// Mitsubishi GX Works2 project: PLC_Group2   PLC: FX3G

// global labels: Global1
VAR_GLOBAL
  StartDay AT X007 : BOOL;
  EmergencyButton AT X011 : BOOL;
  SystemOnLight AT Y007 : BOOL;
  YeastStartValue AT D1160 : INT;
  YeastStock AT D1100 : INT;
  MaltStartValue AT D1170 : INT;
  MaltStock AT D1120 : INT;
  HopsStartValue AT D1180 : INT;
  HopsStock AT D1130 : INT;
  StartCooking AT X001 : BOOL;
  BeerTypeNumber AT D1140 : INT;
END_VAR
VAR_GLOBAL CONSTANT
  Const_5 : INT := 5;
END_VAR
VAR_GLOBAL
  LagerChosen AT M1 : BOOL;
END_VAR
VAR_GLOBAL CONSTANT
  Const_6 : INT := 6;
END_VAR
VAR_GLOBAL
  PilsnerChosen AT M2 : BOOL;
END_VAR
VAR_GLOBAL CONSTANT
  Const_400 : INT := 400;
  Const_150 : INT := 150;
  Const_12 : INT := 12;
  Const_60 : INT := 60;
END_VAR
VAR_GLOBAL
  LagerStockExists AT M3 : BOOL;
END_VAR
VAR_GLOBAL CONSTANT
  Const_120 : INT := 120;
  Const_53 : INT := 53;
END_VAR
VAR_GLOBAL
  PilsnerStockExists AT M4 : BOOL;
END_VAR
VAR_GLOBAL CONSTANT
  Const_4 : INT := 4;
END_VAR
VAR_GLOBAL
  CookingLight AT Y001 : BOOL;
END_VAR
VAR_GLOBAL CONSTANT
  Const_4_Seconds : INT := 40;
END_VAR
VAR_GLOBAL
  CookingTimeIsOver AT TS0 : BOOL;
  CookingTime AT TC0 : BOOL;
  BeerTypeInput AT D8280 : INT;
  StartFermentation AT X005 : BOOL;
  LagerFermentationTimer AT TC1 : BOOL;
  PilsnerFermentationTimer AT TC2 : BOOL;
  Lager_F_TimerIsOver AT TS1 : BOOL;
  Pilsner_F_TimerIsOver AT TS2 : BOOL;
  FermentationIsOver AT M5 : BOOL;
  BlinkingLight1 AT TC3 : BOOL;
  BlinkingLight2 AT TC4 : BOOL;
  BlinkingLight2IsOver AT TS4 : BOOL;
  BlinkingHelp AT M6 : BOOL;
  BlinkingLight1IsOver AT TS3 : BOOL;
  BlinkingLightBall1 AT Y003 : BOOL;
  BlinkingLightBall2 AT Y004 : BOOL;
END_VAR
VAR_GLOBAL CONSTANT
  Const_Half_Second : INT := 5;
END_VAR
VAR_GLOBAL
  StartPacking AT X002 : BOOL;
  Count6Bottles AT CC1 : BOOL;
END_VAR
VAR_GLOBAL CONSTANT
  Counter_6 : INT := 6;
END_VAR
VAR_GLOBAL
  PackBottle AT X000 : BOOL;
  Finished6Bottles AT CS1 : BOOL;
  PackingLight AT Y002 : BOOL;
  TotalPacks AT D1150 : INT;
END_VAR
VAR_GLOBAL CONSTANT
  Const_1 : INT := 1;
END_VAR
VAR_GLOBAL
  NoStock AT M7 : BOOL;
  AnalogOutput AT D8282 : INT;
  GotLagerYeast AT M8 : BOOL;
  GotLagerMalt AT M9 : BOOL;
  GotLagerHops AT M10 : BOOL;
  GotPilsnerYeast AT M11 : BOOL;
  GotPilsnerMalt AT M12 : BOOL;
  GotPilsnerHops AT M13 : BOOL;
END_VAR
VAR_GLOBAL CONSTANT
  Const_40 : INT := 40;
  Const_0 : INT;
END_VAR

// task Task_01 (event TRUE, interval 0, priority 31): POU_01

PROGRAM POU_01
VAR
  TS00 : BOOL;
  TC0 : BOOL;
END_VAR
VAR CONSTANT
  Const_3_Seconds : INT := 30;
  Const_10 : REAL := -10;
END_VAR
(* structured ladder/FBD written out as ST: instructions are called as NAME(EN, inputs, outputs); _pN, _eN, _tN stand for wires *)
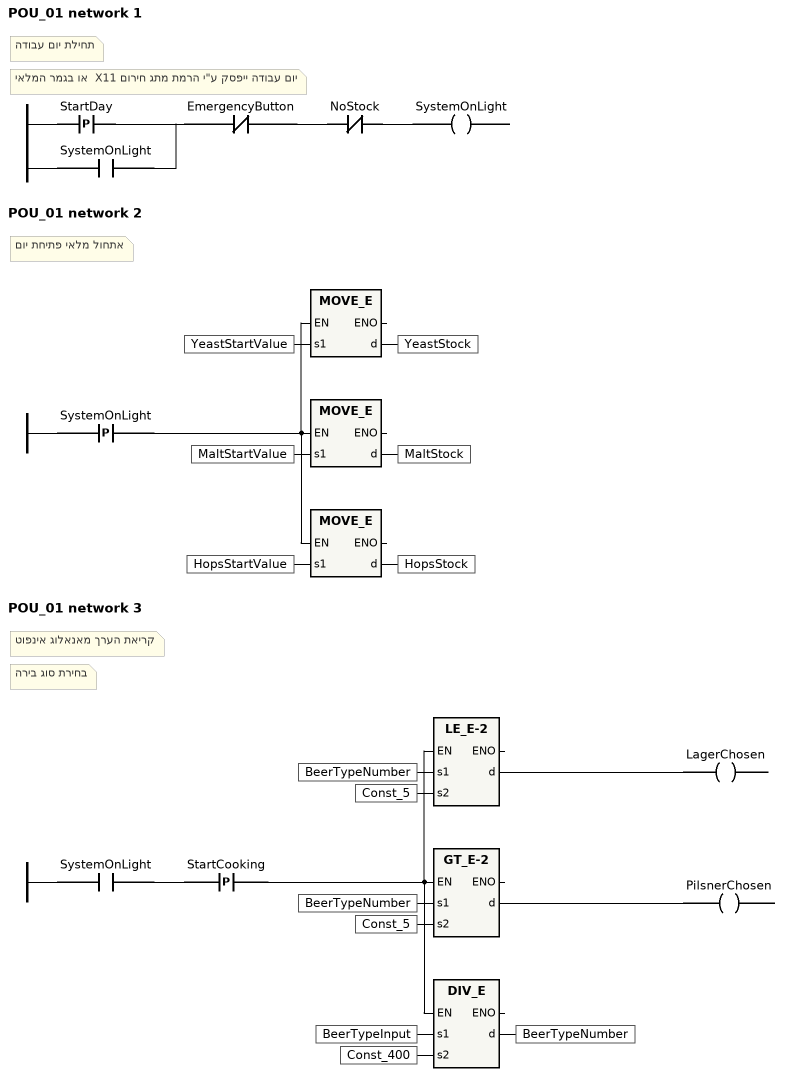
(* network 1 *)
(* תחילת יום עבודה *)
(* יום עבודה ייפסק ע"י הרמת מתג חירום X11  או בגמר המלאי *)
SystemOnLight := ((LDP(TRUE, StartDay) OR SystemOnLight) AND NOT EmergencyButton) AND NOT NoStock;
(* network 2 *)
(* אתחול מלאי פתיחת יום *)
_p1 := LDP(TRUE, SystemOnLight);
MOVE_E(_p1, YeastStartValue, YeastStock);
MOVE_E(_p1, MaltStartValue, MaltStock);
MOVE_E(_p1, HopsStartValue, HopsStock);
(* network 3 *)
(* קריאת הערך מאנאלוג אינפוט *)
(* בחירת סוג בירה *)
_p1 := SystemOnLight AND LDP(TRUE, StartCooking);
DIV_E(_p1, BeerTypeInput, Const_400, BeerTypeNumber);
LE_E(_p1, BeerTypeNumber, Const_5, _t2);
LagerChosen := _t2;
GT_E(_p1, BeerTypeNumber, Const_5, _t3);
PilsnerChosen := _t3;
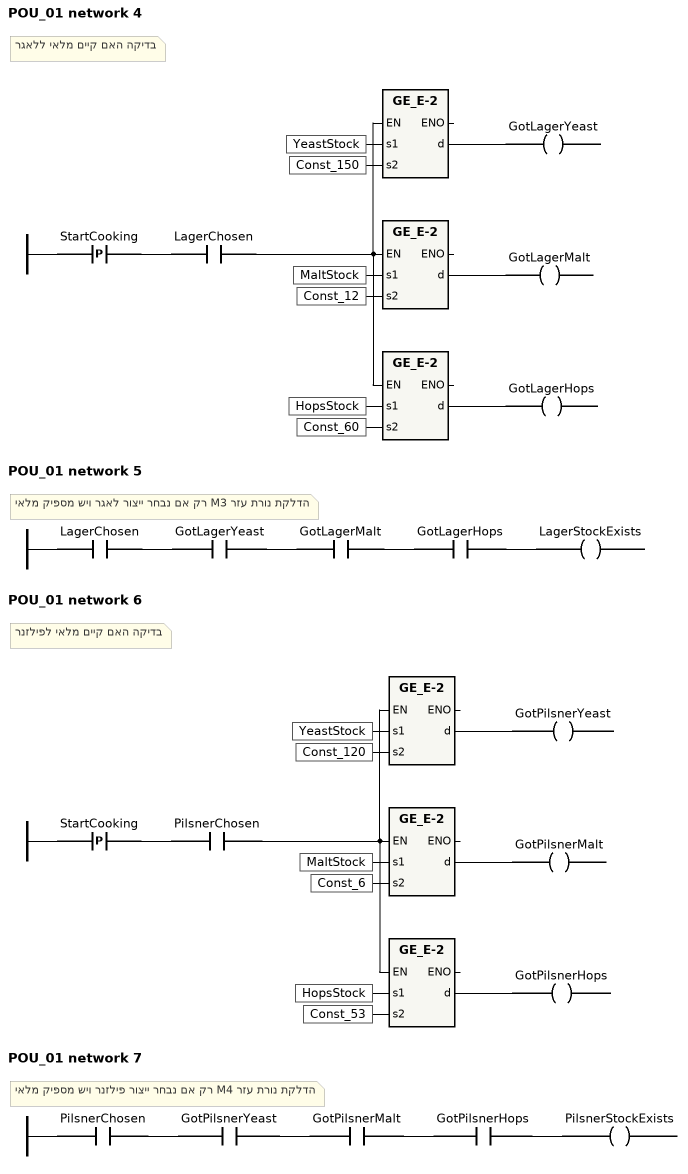
(* network 4 *)
(* בדיקה האם קיים מלאי ללאגר *)
_p1 := LDP(TRUE, StartCooking) AND LagerChosen;
GE_E(_p1, YeastStock, Const_150, _t2);
GotLagerYeast := _t2;
GE_E(_p1, MaltStock, Const_12, _t3);
GotLagerMalt := _t3;
GE_E(_p1, HopsStock, Const_60, _t4);
GotLagerHops := _t4;
(* network 5 *)
(* הדלקת נורת עזר M3 רק אם נבחר ייצור לאגר ויש מספיק מלאי *)
LagerStockExists := LagerChosen AND GotLagerYeast AND GotLagerMalt AND GotLagerHops;
(* network 6 *)
(* בדיקה האם קיים מלאי לפילזנר *)
_p1 := LDP(TRUE, StartCooking) AND PilsnerChosen;
GE_E(_p1, YeastStock, Const_120, _t2);
GotPilsnerYeast := _t2;
GE_E(_p1, MaltStock, Const_6, _t3);
GotPilsnerMalt := _t3;
GE_E(_p1, HopsStock, Const_53, _t4);
GotPilsnerHops := _t4;
(* network 7 *)
(* הדלקת נורת עזר M4 רק אם נבחר ייצור פילזנר ויש מספיק מלאי *)
PilsnerStockExists := PilsnerChosen AND GotPilsnerYeast AND GotPilsnerMalt AND GotPilsnerHops;
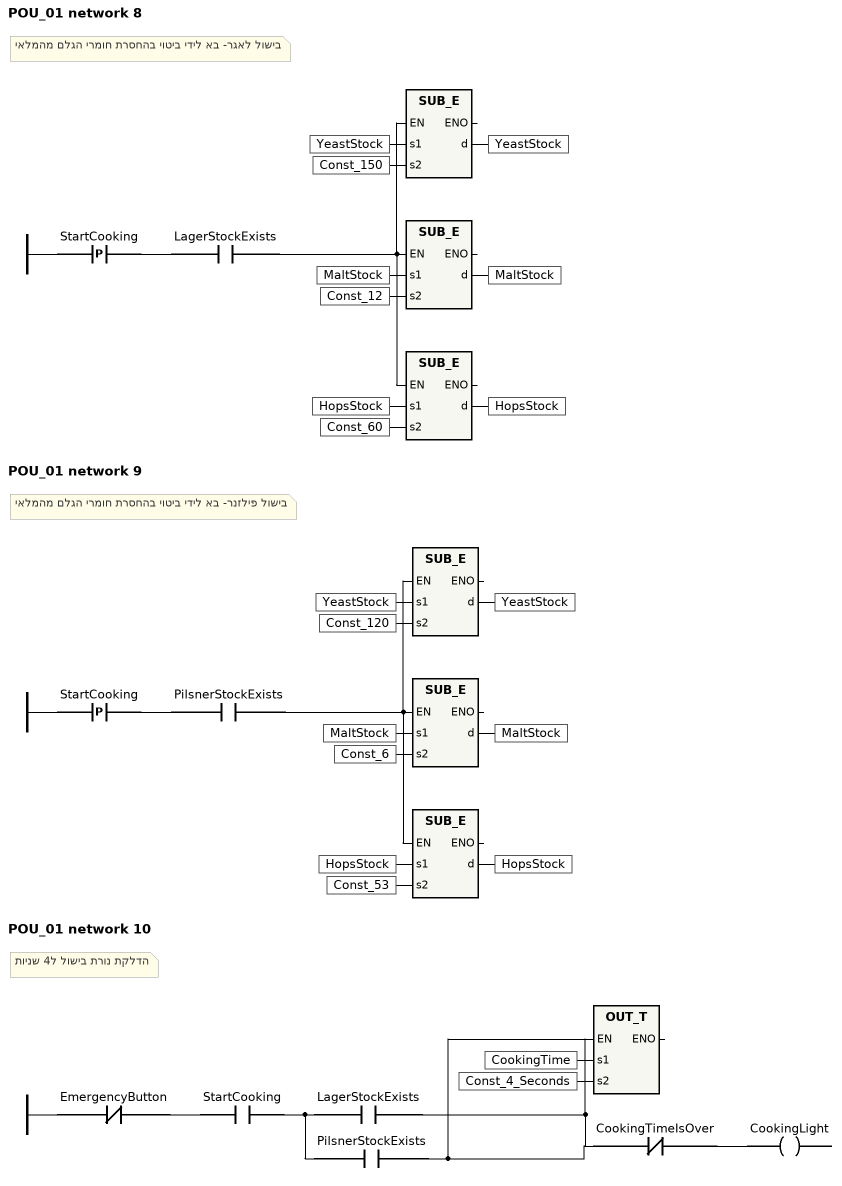
(* network 8 *)
(* בישול לאגר- בא לידי ביטוי בהחסרת חומרי הגלם מהמלאי *)
_p1 := LDP(TRUE, StartCooking) AND LagerStockExists;
SUB_E(_p1, YeastStock, Const_150, YeastStock);
SUB_E(_p1, MaltStock, Const_12, MaltStock);
SUB_E(_p1, HopsStock, Const_60, HopsStock);
(* network 9 *)
(* בישול פילזנר- בא לידי ביטוי בהחסרת חומרי הגלם מהמלאי *)
_p1 := LDP(TRUE, StartCooking) AND PilsnerStockExists;
SUB_E(_p1, YeastStock, Const_120, YeastStock);
SUB_E(_p1, MaltStock, Const_6, MaltStock);
SUB_E(_p1, HopsStock, Const_53, HopsStock);
(* network 10 *)
(* הדלקת נורת בישול ל4 שניות *)
_p1 := NOT EmergencyButton AND StartCooking;
_p2 := (_p1 AND LagerStockExists) OR (_p1 AND PilsnerStockExists);
OUT_T(_p2, CookingTime, Const_4_Seconds);
CookingLight := _p2 AND NOT CookingTimeIsOver;
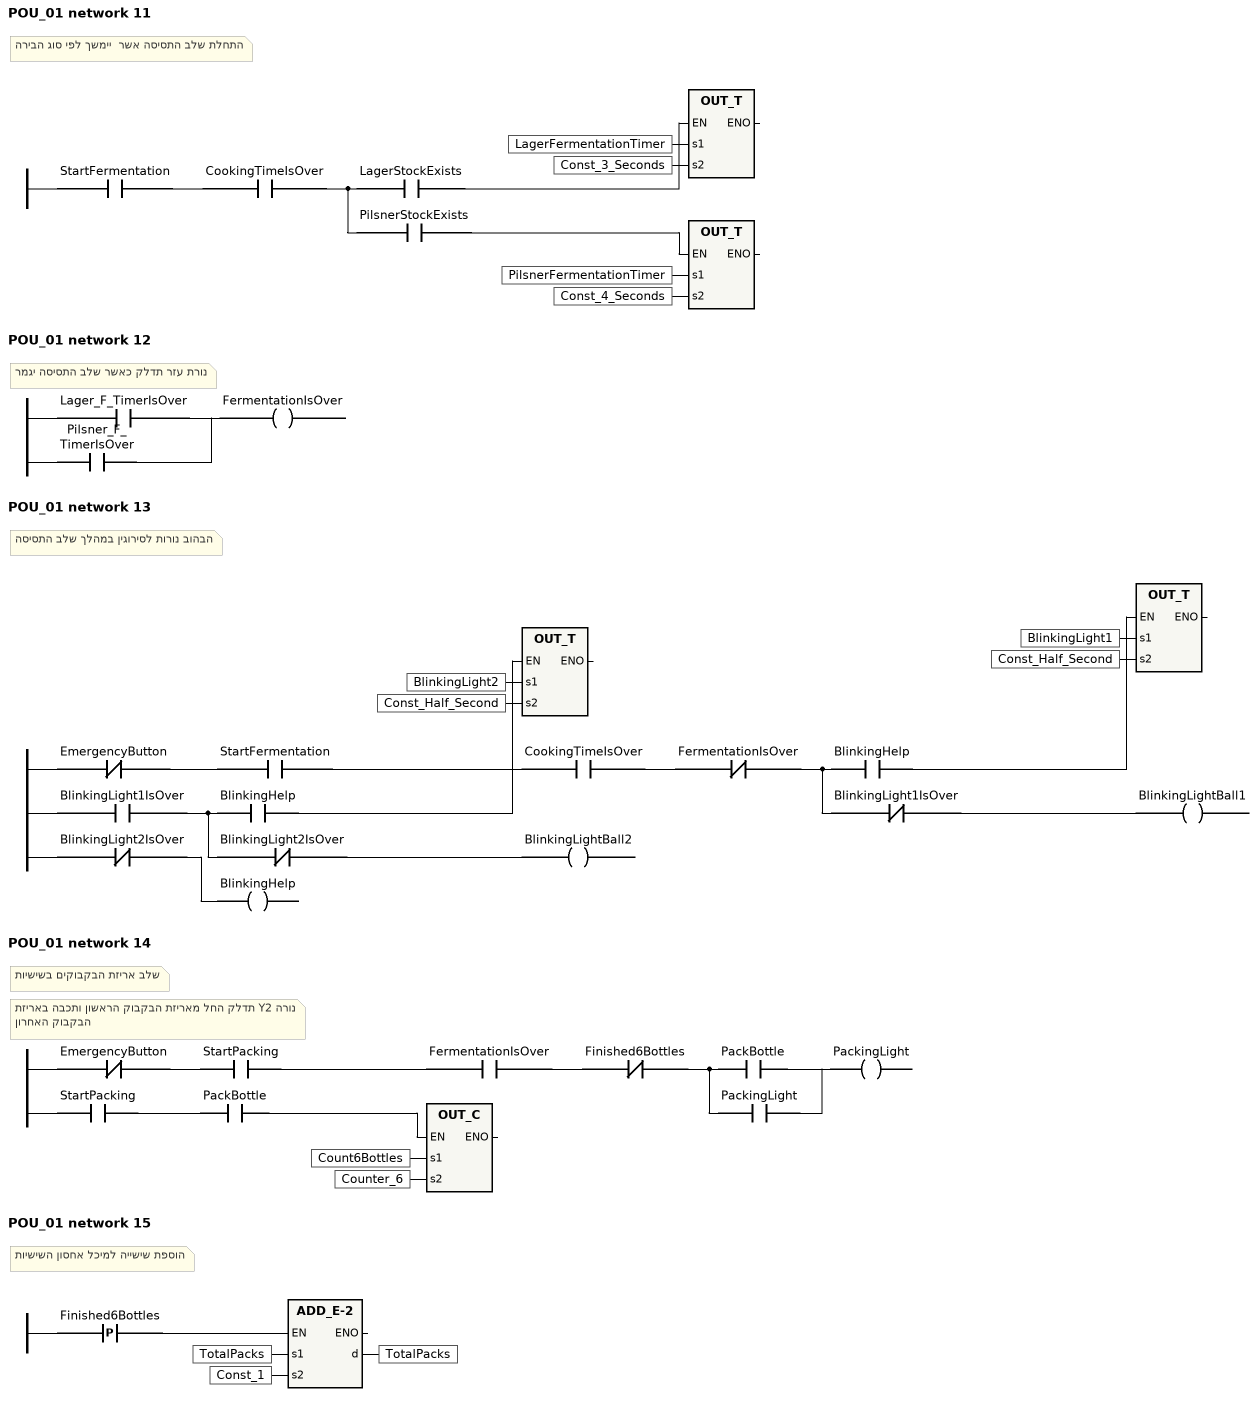
(* network 11 *)
(* התחלת שלב התסיסה אשר  יימשך לפי סוג הבירה *)
_p1 := StartFermentation AND CookingTimeIsOver;
OUT_T(_p1 AND LagerStockExists, LagerFermentationTimer, Const_3_Seconds);
OUT_T(_p1 AND PilsnerStockExists, PilsnerFermentationTimer, Const_4_Seconds);
(* network 12 *)
(* נורת עזר תדלק כאשר שלב התסיסה יגמר *)
FermentationIsOver := Lager_F_TimerIsOver OR Pilsner_F_TimerIsOver;
(* network 13 *)
(* הבהוב נורות לסירוגין במהלך שלב התסיסה *)
_p1 := NOT EmergencyButton AND StartFermentation AND CookingTimeIsOver AND NOT FermentationIsOver;
OUT_T(_p1 AND BlinkingHelp, BlinkingLight1, Const_Half_Second);
BlinkingLightBall1 := _p1 AND NOT BlinkingLight1IsOver;
OUT_T(BlinkingLight1IsOver AND BlinkingHelp, BlinkingLight2, Const_Half_Second);
BlinkingLightBall2 := BlinkingLight1IsOver AND NOT BlinkingLight2IsOver;
BlinkingHelp := NOT BlinkingLight2IsOver;
(* network 14 *)
(* שלב אריזת הבקבוקים בשישיות *)
(* נורה Y2 תדלק החל מאריזת הבקבוק הראשון ותכבה באריזת הבקבוק האחרון *)
_p1 := NOT EmergencyButton AND StartPacking AND FermentationIsOver AND NOT Finished6Bottles;
PackingLight := (_p1 AND PackBottle) OR (_p1 AND PackingLight);
OUT_C(StartPacking AND PackBottle, Count6Bottles, Counter_6);
(* network 15 *)
(* הוספת שישייה למיכל אחסון השישיות *)
ADD_E(LDP(TRUE, Finished6Bottles), TotalPacks, Const_1, TotalPacks);
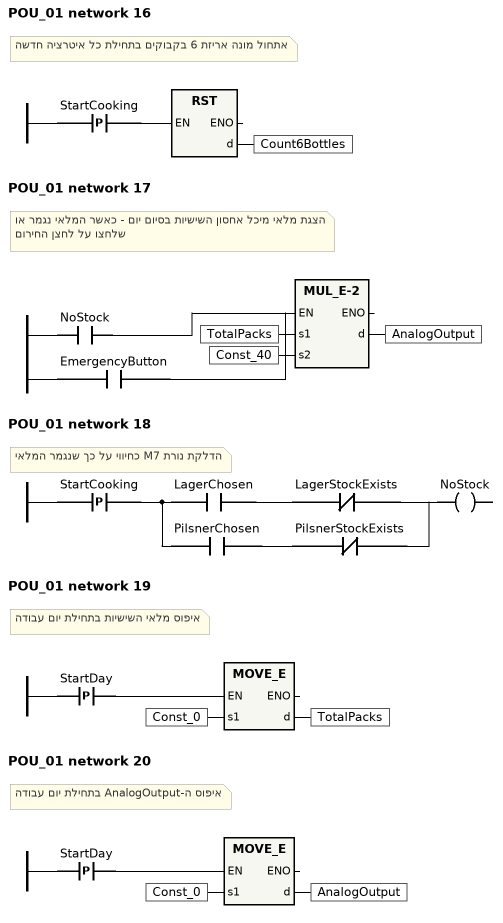
(* network 16 *)
(* אתחול מונה אריזת 6 בקבוקים בתחילת כל איטרציה חדשה *)
RST(LDP(TRUE, StartCooking), Count6Bottles);
(* network 17 *)
(* הצגת מלאי מיכל אחסון השישיות בסיום יום - כאשר המלאי נגמר או שלחצו על לחצן החירום *)
MUL_E(NoStock OR EmergencyButton, TotalPacks, Const_40, AnalogOutput);
(* network 18 *)
(* הדלקת נורת M7 כחיווי על כך שנגמר המלאי *)
_p1 := LDP(TRUE, StartCooking);
NoStock := (_p1 AND LagerChosen AND NOT LagerStockExists) OR (_p1 AND PilsnerChosen AND NOT PilsnerStockExists);
(* network 19 *)
(* איפוס מלאי השישיות בתחילת יום עבודה *)
MOVE_E(LDP(TRUE, StartDay), Const_0, TotalPacks);
(* network 20 *)
(* איפוס ה-AnalogOutput בתחילת יום עבודה *)
MOVE_E(LDP(TRUE, StartDay), Const_0, AnalogOutput);
END_PROGRAM
